Omron Sysmac Studio project FileStreamReader (Sysmac Studio 1.60.0.10, StandardProject)
(* CASEステートマシンの使用例。 *)

# Controller Example: NX102-1000 version 1.64
Task PrimaryTask (priority 4, period or condition 2000): Main

TYPE StreamContext : STRUCT
    Buffer : ARRAY[0..65534] OF BYTE;
    Head : UINT;
    Tail : UINT;
    Size : UINT;
    End : BOOL;
    ReadSize : UDINT;
    WriteSize : UDINT;
    Error : BOOL;
    ErrorID : WORD;
    ErrorIDEx : DWORD;
END_STRUCT END_TYPE

PROGRAM Main
VAR
    iState : UINT;
    iFileReader : FileStreamReader;
    iContext : StreamContext;
    iBuffer : ARRAY[0..127] OF BYTE;
    iReadSize : UINT;
    iMessage : STRING[256];
    iWaitTick : UINT;
    iErrorID : WORD;
    iErrorIDEx : DWORD;
END_VAR
(*
 * ファイルストリームリーダー使用例
 *
 * [使い方]
 * 1. "C:\OMRON\Data\SimulatorData\CARD\Memory001"にASCII文字列の適当なファイルを入れます。
 * 2. "iFileReader.Path"にファイルパス(仮想SD内にあるとして)を指定します。
 * 3. シミュレータを実行します。
 *
 * © 2024 KITA Munemitsu
 *)
 
CASE iState OF
	// ファイルリーダー初期化
	0:
		iFileReader.Execute := FALSE;
		
		Inc(iState);
	1:
	 	// 99999文字のLorem ipsumのファイルです。POU/プログラム/loremipsumのコメント内にコンテンツがあります。
		iFileReader.Path := '/loremipsum.txt';
		
		//"0"が65533文字、"1"が1文字のファイルです。POU/プログラム/zero_65533_one_1のコメント内にコンテンツがあります。
		// iFileReader.Path := '/zero_65533_one_1.txt';
		
		//"0"が65534文字、"1"が1文字のファイルです。POU/プログラム/zero_65534_one_1のコメント内にコンテンツがあります。
		// iFileReader.Path := '/zero_65534_one_1.txt';
		
		//"0"が65535文字、"1"が1文字のファイルです。POU/プログラム/zero_65535_one_1のコメント内にコンテンツがあります。
		// iFileReader.Path := '/zero_65535_one_1.txt';
		
		iFileReader.Execute := TRUE;
				
		Inc(iState);
		
	// ストリーム処理
	2:
		// ストリームでエラーが発生したら実行します。
		IF Stream_OnError(Context:=iContext) THEN
			iMessage := 'Fatal error...';
			Stream_ErrorInfo(Context:=iContext, ErrorID=>iErrorID, ErrorIDEx=>iErrorIDEx);
			
			iState := iState + 7;
		// ストリームが終了すると実行します。
		ELSIF Stream_OnEnd(Context:=iContext) THEN
			iMessage := 'Done!!';
			
			iState := iState + 7;
		// ストリームにデータが存在したら実行します。
		ELSIF Stream_OnData(
			   Context:=iContext,
			   Out:=iBuffer,
			   OutHead:=0,
			   OutSize=>iReadSize)
		THEN
			iMessage := AryToString(In:=iBuffer[0], Size:=iReadSize);
			iWaitTick := 10;
			
			Inc(iState);
		END_IF;
	3: // ストリーム処理に必要ではありませんが、無いとすぐに終了してしまいます。
		Dec(iWaitTick);
		IF iWaitTick < 1 THEN
			Dec(iState);
		END_IF;
	
	// ストリーム処理終了
	9:
		iFileReader.Execute := FALSE;
		
		Inc(iState);
END_CASE;

iFileReader(Context:=iContext);
END_PROGRAM

PROGRAM README
RETURN;
(*
このプロジェクトは、CASEステートマシンの事例として作成したものです。
CASEステートマシンが効果を発揮する非同期FBの使用例として、
SDカード命令を使用し、ファイル読み出しをストリーム化します。
学習用途には十分ですが、実使用に耐えるものではありません。

POU/ファンクションブロック/FileStreamReaderがストリーム処理を実行するFBです。
POU/Stream_OnData、Stream_OnEnd、Stream_OnError、Stream_ErrorInfoはストリームを使用するためのFUNです。
POU/プログラム/Mainが使用例のプログラムです。

私に権利のある部分については、POU/LICENSEに従います。
使用、改変は自由ですがそれに係る一切の損害・損失の責任は負いません。
*)
END_PROGRAM

PROGRAM LICENSE
RETURN;
(*
The MIT License (MIT)

Copyright(c) 2024 KITA Munemitsu

Permission is hereby granted, free of charge, to any person obtaining a copy of this software and associated
documentation files (the “Software”), to deal in the Software without restriction, including without limitation
the rights to use, copy, modify, merge, publish, distribute, sublicense, and/or sell copies of the Software,
and to permit persons to whom the Software is furnished to do so, subject to the following conditions:

The above copyright notice and this permission notice shall be included in all copies or substantial portions of the Software.

THE SOFTWARE IS PROVIDED “AS IS”, WITHOUT WARRANTY OF ANY KIND, EXPRESS OR IMPLIED, INCLUDING BUT NOT
LIMITED TO THE WARRANTIES OF MERCHANTABILITY, FITNESS FOR A PARTICULAR PURPOSE AND NONINFRINGEMENT.
IN NO EVENT SHALL THE AUTHORS OR COPYRIGHT HOLDERS BE LIABLE FOR ANY CLAIM, DAMAGES OR OTHER LIABILITY,
WHETHER IN AN ACTION OF CONTRACT, TORT OR OTHERWISE, ARISING FROM, OUT OF OR IN CONNECTION WITH THE SOFTWARE
OR THE USE OR OTHER DEALINGS IN THE SOFTWARE.
*)
END_PROGRAM

PROGRAM loremipsum
RETURN;
(* loremipsum.txt
